{attribute 'GeneratedUsingTerminal: CX1100-0004-0000'}
{attribute addProperty BoxType "CX1100-0004-0000"}
{attribute addProperty Id "InfoDataAT %I*InfoData_6F19DB2B2"}
{attribute addProperty CRC "532711307"}
{attribute addProperty Size "2"}
TYPE CX1100_1FC0878B EXTENDS EtcSlaveTerminalBase_947E5A46 :
STRUCT
	{attribute addProperty Name "InfoData"}
	InfoData : InfoData_6F19DB2B;
END_STRUCT
END_TYPE

(* stored: Version 1.2.0.0, ProductVersion 3.1.4024.9
   DUT CX1100_1FC0878B: Id {d4068f95-233f-4c64-9dd2-eb0fb9f1cc4f} *)
